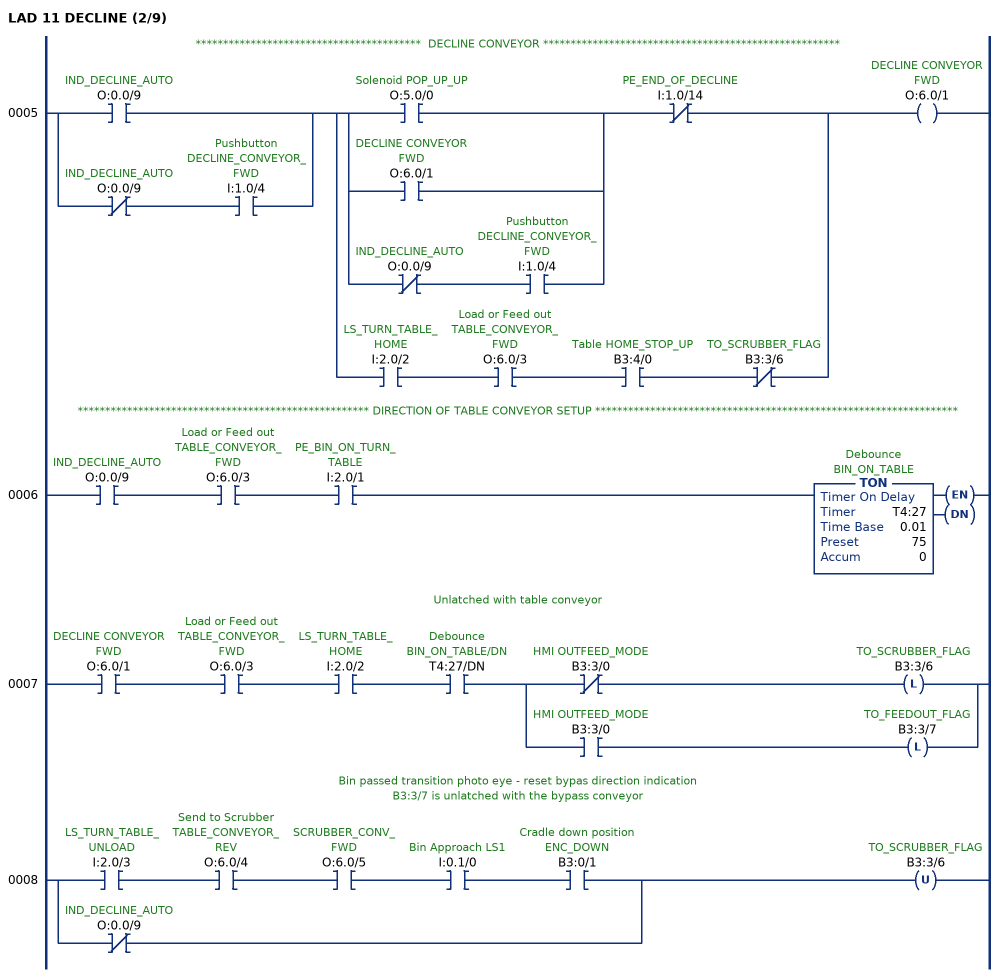
% Rung: 5 %
% *****************************************  DECLINE CONVEYOR ****************************************************** %
SOR BST XIC O:0.0/9 NXB XIO O:0.0/9 XIC I:1.0/4 BND BST BST XIC O:5.0/0 NXB BST XIC O:6.0/1 NXB XIO O:0.0/9 XIC I:1.0/4 BND BND XIO I:1.0/14 NXB XIC I:2.0/2 XIC O:6.0/3 XIC B3:4/0 XIO B3:3/6 BND OTE O:6.0/1 EOR
%   O:0.0/9  IND_DECLINE_AUTO %
%   I:1.0/4  DECLINE_CONVEYOR_FWD  "Pushbutton" %
%   O:5.0/0  POP_UP_UP  "Solenoid" %
%   O:6.0/1  "DECLINE CONVEYOR FWD" %
%   I:1.0/14  PE_END_OF_DECLINE %
%   I:2.0/2  LS_TURN_TABLE_HOME %
%   O:6.0/3  TABLE_CONVEYOR_FWD  "Load or Feed out" %
%   B3:4/0  HOME_STOP_UP  "Table" %
%   B3:3/6  TO_SCRUBBER_FLAG %
% Rung: 6 %
% ***************************************************** DIRECTION OF TABLE CONVEYOR SETUP ****************************************************************** %
SOR XIC O:0.0/9 XIC O:6.0/3 XIC I:2.0/1 TON T4:27 0.01 75 0 EOR
%   O:0.0/9  IND_DECLINE_AUTO %
%   O:6.0/3  TABLE_CONVEYOR_FWD  "Load or Feed out" %
%   I:2.0/1  PE_BIN_ON_TURN_TABLE %
%   T4:27  BIN_ON_TABLE  "Debounce" %
% Rung: 7 %
% Unlatched with table conveyor %
SOR XIC O:6.0/1 XIC O:6.0/3 XIC I:2.0/2 XIC T4:27/DN BST XIO B3:3/0 OTL B3:3/6 NXB XIC B3:3/0 OTL B3:3/7 BND EOR
%   O:6.0/1  "DECLINE CONVEYOR FWD" %
%   O:6.0/3  TABLE_CONVEYOR_FWD  "Load or Feed out" %
%   I:2.0/2  LS_TURN_TABLE_HOME %
%   T4:27  BIN_ON_TABLE  "Debounce" %
%   B3:3/0  OUTFEED_MODE  "HMI" %
%   B3:3/6  TO_SCRUBBER_FLAG %
%   B3:3/7  TO_FEEDOUT_FLAG %
% Rung: 8 %
% Bin passed transition photo eye - reset bypas direction indication
% B3:3/7 is unlatched with the bypass conveyor %
SOR BST XIC I:2.0/3 XIC O:6.0/4 XIC O:6.0/5 XIC I:0.1/0 XIC B3:0/1 NXB XIO O:0.0/9 BND OTU B3:3/6 EOR
%   I:2.0/3  LS_TURN_TABLE_UNLOAD %
%   O:6.0/4  TABLE_CONVEYOR_REV  "Send to Scrubber" %
%   O:6.0/5  SCRUBBER_CONV_FWD %
%   I:0.1/0  LS1  "Bin Approach" %
%   B3:0/1  ENC_DOWN  "Cradle down position" %
%   O:0.0/9  IND_DECLINE_AUTO %
%   B3:3/6  TO_SCRUBBER_FLAG %

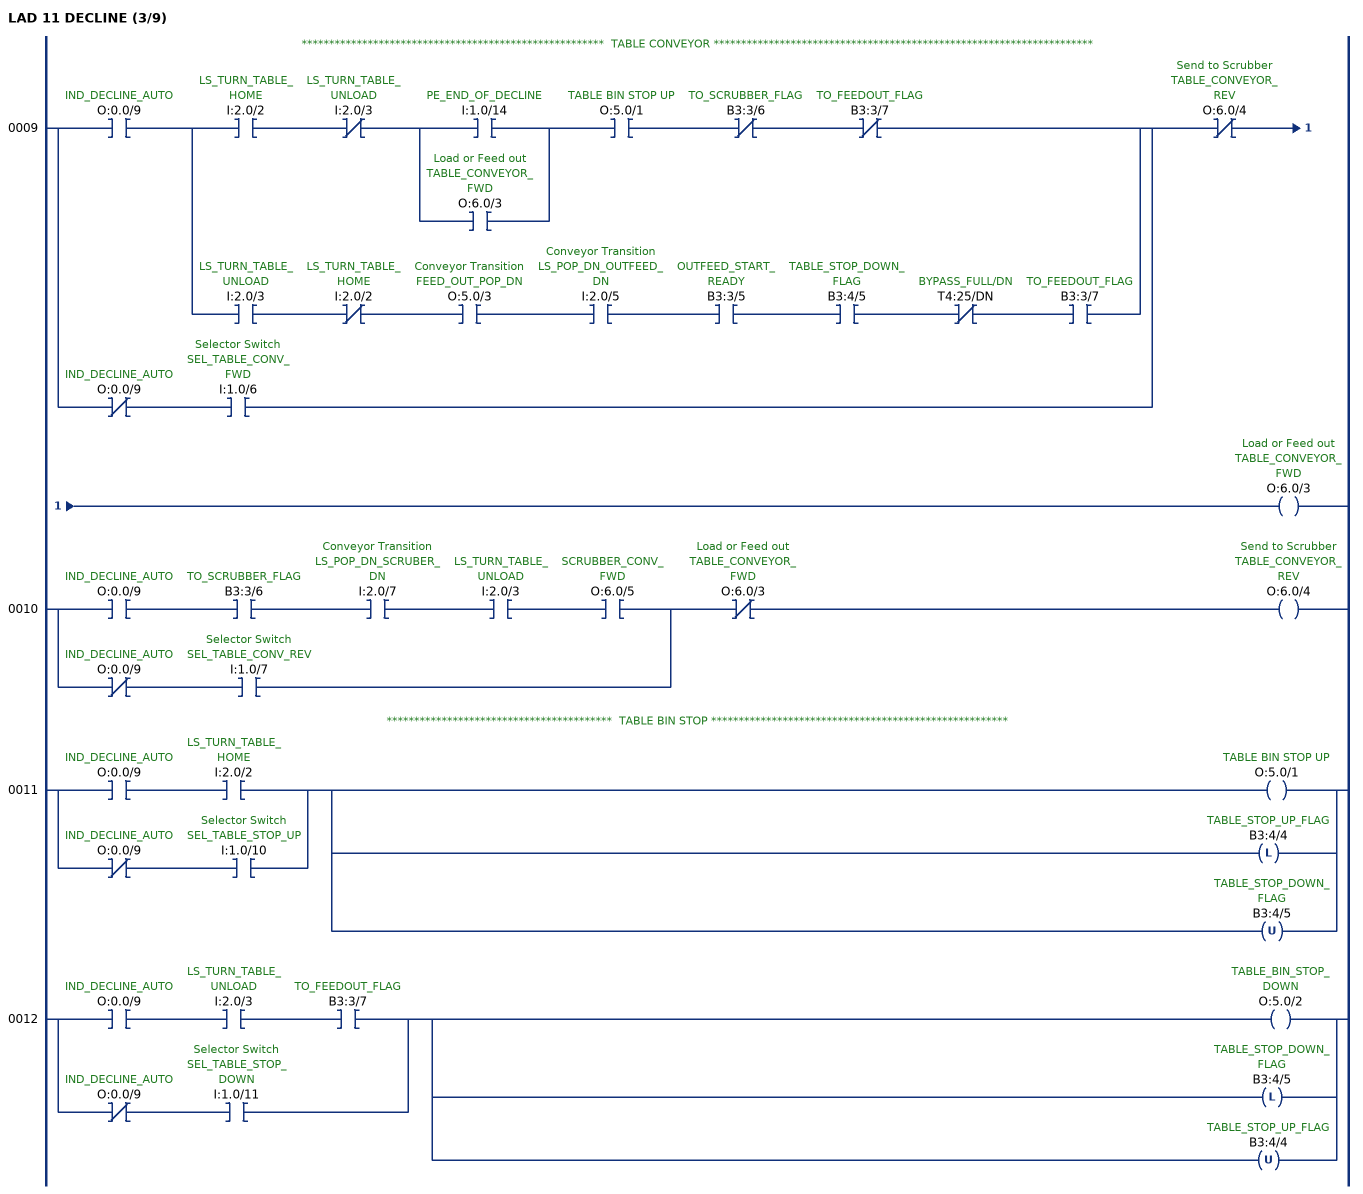
% Rung: 9 %
% *******************************************************  TABLE CONVEYOR ********************************************************************* %
SOR BST XIC O:0.0/9 BST XIC I:2.0/2 XIO I:2.0/3 BST XIC I:1.0/14 NXB XIC O:6.0/3 BND XIC O:5.0/1 XIO B3:3/6 XIO B3:3/7 NXB XIC I:2.0/3 XIO I:2.0/2 XIC O:5.0/3 XIC I:2.0/5 XIC B3:3/5 XIC B3:4/5 XIO T4:25/DN XIC B3:3/7 BND NXB XIO O:0.0/9 XIC I:1.0/6 BND XIO O:6.0/4 OTE O:6.0/3 EOR
%   O:0.0/9  IND_DECLINE_AUTO %
%   I:2.0/2  LS_TURN_TABLE_HOME %
%   I:2.0/3  LS_TURN_TABLE_UNLOAD %
%   I:1.0/14  PE_END_OF_DECLINE %
%   O:6.0/3  TABLE_CONVEYOR_FWD  "Load or Feed out" %
%   O:5.0/1  "TABLE BIN STOP UP" %
%   B3:3/6  TO_SCRUBBER_FLAG %
%   B3:3/7  TO_FEEDOUT_FLAG %
%   O:5.0/3  FEED_OUT_POP_DN  "Conveyor Transition" %
%   I:2.0/5  LS_POP_DN_OUTFEED_DN  "Conveyor Transition" %
%   B3:3/5  OUTFEED_START_READY %
%   B3:4/5  TABLE_STOP_DOWN_FLAG %
%   T4:25  BYPASS_FULL %
%   I:1.0/6  SEL_TABLE_CONV_FWD  "Selector Switch" %
%   O:6.0/4  TABLE_CONVEYOR_REV  "Send to Scrubber" %
% Rung: 10 %
SOR BST XIC O:0.0/9 XIC B3:3/6 XIC I:2.0/7 XIC I:2.0/3 XIC O:6.0/5 NXB XIO O:0.0/9 XIC I:1.0/7 BND XIO O:6.0/3 OTE O:6.0/4 EOR
%   O:0.0/9  IND_DECLINE_AUTO %
%   B3:3/6  TO_SCRUBBER_FLAG %
%   I:2.0/7  LS_POP_DN_SCRUBER_DN  "Conveyor Transition" %
%   I:2.0/3  LS_TURN_TABLE_UNLOAD %
%   O:6.0/5  SCRUBBER_CONV_FWD %
%   I:1.0/7  SEL_TABLE_CONV_REV  "Selector Switch" %
%   O:6.0/3  TABLE_CONVEYOR_FWD  "Load or Feed out" %
%   O:6.0/4  TABLE_CONVEYOR_REV  "Send to Scrubber" %
% Rung: 11 %
% *****************************************  TABLE BIN STOP ****************************************************** %
SOR BST XIC O:0.0/9 XIC I:2.0/2 NXB XIO O:0.0/9 XIC I:1.0/10 BND BST OTE O:5.0/1 NXB BST OTL B3:4/4 NXB OTU B3:4/5 BND BND EOR
%   O:0.0/9  IND_DECLINE_AUTO %
%   I:2.0/2  LS_TURN_TABLE_HOME %
%   I:1.0/10  SEL_TABLE_STOP_UP  "Selector Switch" %
%   O:5.0/1  "TABLE BIN STOP UP" %
%   B3:4/4  TABLE_STOP_UP_FLAG %
%   B3:4/5  TABLE_STOP_DOWN_FLAG %
% Rung: 12 %
SOR BST XIC O:0.0/9 XIC I:2.0/3 XIC B3:3/7 NXB XIO O:0.0/9 XIC I:1.0/11 BND BST OTE O:5.0/2 NXB BST OTL B3:4/5 NXB OTU B3:4/4 BND BND EOR
%   O:0.0/9  IND_DECLINE_AUTO %
%   I:2.0/3  LS_TURN_TABLE_UNLOAD %
%   B3:3/7  TO_FEEDOUT_FLAG %
%   I:1.0/11  SEL_TABLE_STOP_DOWN  "Selector Switch" %
%   O:5.0/2  "TABLE_BIN_STOP_DOWN" %
%   B3:4/5  TABLE_STOP_DOWN_FLAG %
%   B3:4/4  TABLE_STOP_UP_FLAG %

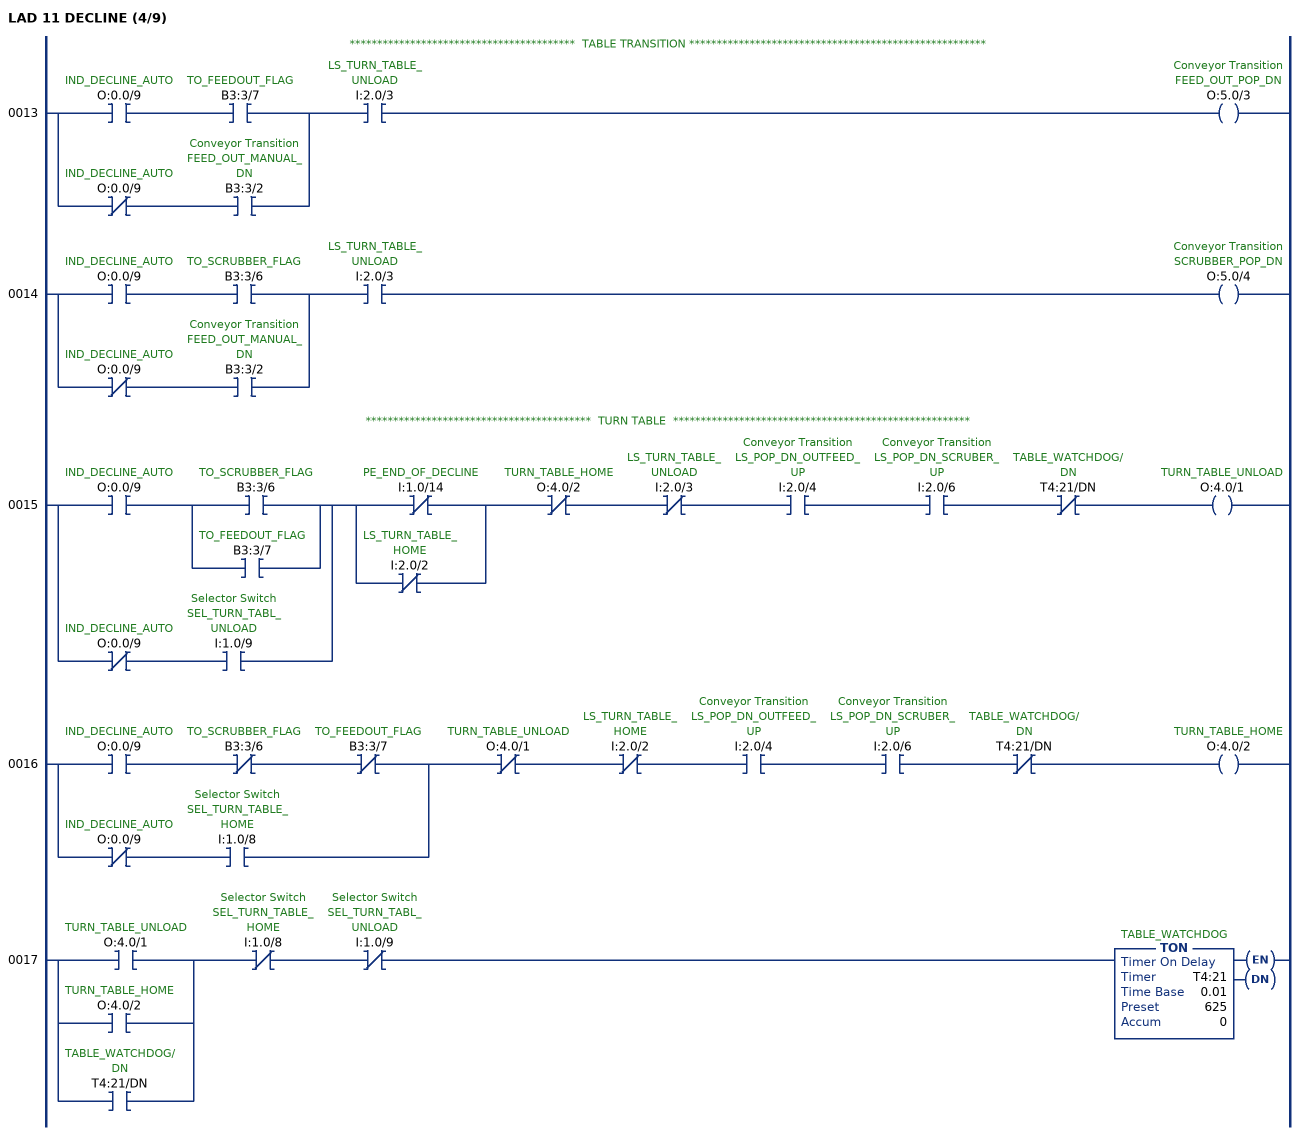
% Rung: 13 %
% *****************************************  TABLE TRANSITION ****************************************************** %
SOR BST XIC O:0.0/9 XIC B3:3/7 NXB XIO O:0.0/9 XIC B3:3/2 BND XIC I:2.0/3 OTE O:5.0/3 EOR
%   O:0.0/9  IND_DECLINE_AUTO %
%   B3:3/7  TO_FEEDOUT_FLAG %
%   B3:3/2  FEED_OUT_MANUAL_DN  "Conveyor Transition" %
%   I:2.0/3  LS_TURN_TABLE_UNLOAD %
%   O:5.0/3  FEED_OUT_POP_DN  "Conveyor Transition" %
% Rung: 14 %
SOR BST XIC O:0.0/9 XIC B3:3/6 NXB XIO O:0.0/9 XIC B3:3/2 BND XIC I:2.0/3 OTE O:5.0/4 EOR
%   O:0.0/9  IND_DECLINE_AUTO %
%   B3:3/6  TO_SCRUBBER_FLAG %
%   B3:3/2  FEED_OUT_MANUAL_DN  "Conveyor Transition" %
%   I:2.0/3  LS_TURN_TABLE_UNLOAD %
%   O:5.0/4  SCRUBBER_POP_DN  "Conveyor Transition" %
% Rung: 15 %
% *****************************************  TURN TABLE  ****************************************************** %
SOR BST XIC O:0.0/9 BST XIC B3:3/6 NXB XIC B3:3/7 BND NXB XIO O:0.0/9 XIC I:1.0/9 BND BST XIO I:1.0/14 NXB XIO I:2.0/2 BND XIO O:4.0/2 XIO I:2.0/3 XIC I:2.0/4 XIC I:2.0/6 XIO T4:21/DN OTE O:4.0/1 EOR
%   O:0.0/9  IND_DECLINE_AUTO %
%   B3:3/6  TO_SCRUBBER_FLAG %
%   B3:3/7  TO_FEEDOUT_FLAG %
%   I:1.0/9  SEL_TURN_TABL_UNLOAD  "Selector Switch" %
%   I:1.0/14  PE_END_OF_DECLINE %
%   I:2.0/2  LS_TURN_TABLE_HOME %
%   O:4.0/2  TURN_TABLE_HOME %
%   I:2.0/3  LS_TURN_TABLE_UNLOAD %
%   I:2.0/4  LS_POP_DN_OUTFEED_UP  "Conveyor Transition" %
%   I:2.0/6  LS_POP_DN_SCRUBER_UP  "Conveyor Transition" %
%   T4:21  TABLE_WATCHDOG %
%   O:4.0/1  TURN_TABLE_UNLOAD %
% Rung: 16 %
SOR BST XIC O:0.0/9 XIO B3:3/6 XIO B3:3/7 NXB XIO O:0.0/9 XIC I:1.0/8 BND XIO O:4.0/1 XIO I:2.0/2 XIC I:2.0/4 XIC I:2.0/6 XIO T4:21/DN OTE O:4.0/2 EOR
%   O:0.0/9  IND_DECLINE_AUTO %
%   B3:3/6  TO_SCRUBBER_FLAG %
%   B3:3/7  TO_FEEDOUT_FLAG %
%   I:1.0/8  SEL_TURN_TABLE_HOME  "Selector Switch" %
%   O:4.0/1  TURN_TABLE_UNLOAD %
%   I:2.0/2  LS_TURN_TABLE_HOME %
%   I:2.0/4  LS_POP_DN_OUTFEED_UP  "Conveyor Transition" %
%   I:2.0/6  LS_POP_DN_SCRUBER_UP  "Conveyor Transition" %
%   T4:21  TABLE_WATCHDOG %
%   O:4.0/2  TURN_TABLE_HOME %
% Rung: 17 %
SOR BST BST XIC O:4.0/1 NXB XIC O:4.0/2 BND NXB XIC T4:21/DN BND XIO I:1.0/8 XIO I:1.0/9 TON T4:21 0.01 625 0 EOR
%   O:4.0/1  TURN_TABLE_UNLOAD %
%   O:4.0/2  TURN_TABLE_HOME %
%   T4:21  TABLE_WATCHDOG %
%   I:1.0/8  SEL_TURN_TABLE_HOME  "Selector Switch" %
%   I:1.0/9  SEL_TURN_TABL_UNLOAD  "Selector Switch" %

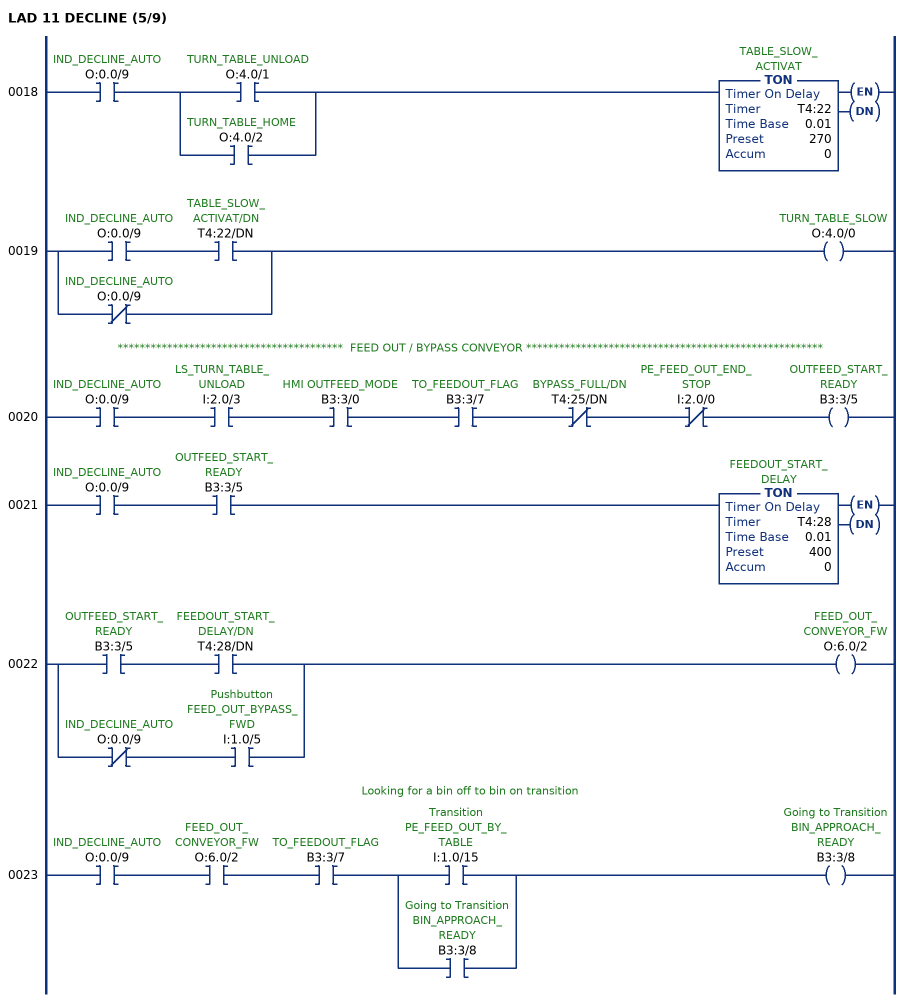
% Rung: 18 %
SOR XIC O:0.0/9 BST XIC O:4.0/1 NXB XIC O:4.0/2 BND TON T4:22 0.01 270 0 EOR
%   O:0.0/9  IND_DECLINE_AUTO %
%   O:4.0/1  TURN_TABLE_UNLOAD %
%   O:4.0/2  TURN_TABLE_HOME %
%   T4:22  TABLE_SLOW_ACTIVAT %
% Rung: 19 %
SOR BST XIC O:0.0/9 XIC T4:22/DN NXB XIO O:0.0/9 BND OTE O:4.0/0 EOR
%   O:0.0/9  IND_DECLINE_AUTO %
%   T4:22  TABLE_SLOW_ACTIVAT %
%   O:4.0/0  TURN_TABLE_SLOW %
% Rung: 20 %
% *****************************************  FEED OUT / BYPASS CONVEYOR ****************************************************** %
SOR XIC O:0.0/9 XIC I:2.0/3 XIC B3:3/0 XIC B3:3/7 XIO T4:25/DN XIO I:2.0/0 OTE B3:3/5 EOR
%   O:0.0/9  IND_DECLINE_AUTO %
%   I:2.0/3  LS_TURN_TABLE_UNLOAD %
%   B3:3/0  OUTFEED_MODE  "HMI" %
%   B3:3/7  TO_FEEDOUT_FLAG %
%   T4:25  BYPASS_FULL %
%   I:2.0/0  PE_FEED_OUT_END_STOP %
%   B3:3/5  OUTFEED_START_READY %
% Rung: 21 %
SOR XIC O:0.0/9 XIC B3:3/5 TON T4:28 0.01 400 0 EOR
%   O:0.0/9  IND_DECLINE_AUTO %
%   B3:3/5  OUTFEED_START_READY %
%   T4:28  FEEDOUT_START_DELAY %
% Rung: 22 %
SOR BST XIC B3:3/5 XIC T4:28/DN NXB XIO O:0.0/9 XIC I:1.0/5 BND OTE O:6.0/2 EOR
%   B3:3/5  OUTFEED_START_READY %
%   T4:28  FEEDOUT_START_DELAY %
%   O:0.0/9  IND_DECLINE_AUTO %
%   I:1.0/5  FEED_OUT_BYPASS_FWD  "Pushbutton" %
%   O:6.0/2  FEED_OUT_CONVEYOR_FW %
% Rung: 23 %
% Looking for a bin off to bin on transition %
SOR XIC O:0.0/9 XIC O:6.0/2 XIC B3:3/7 BST XIC I:1.0/15 NXB XIC B3:3/8 BND OTE B3:3/8 EOR
%   O:0.0/9  IND_DECLINE_AUTO %
%   O:6.0/2  FEED_OUT_CONVEYOR_FW %
%   B3:3/7  TO_FEEDOUT_FLAG %
%   I:1.0/15  PE_FEED_OUT_BY_TABLE  "Transition" %
%   B3:3/8  BIN_APPROACH_READY  "Going to Transition" %

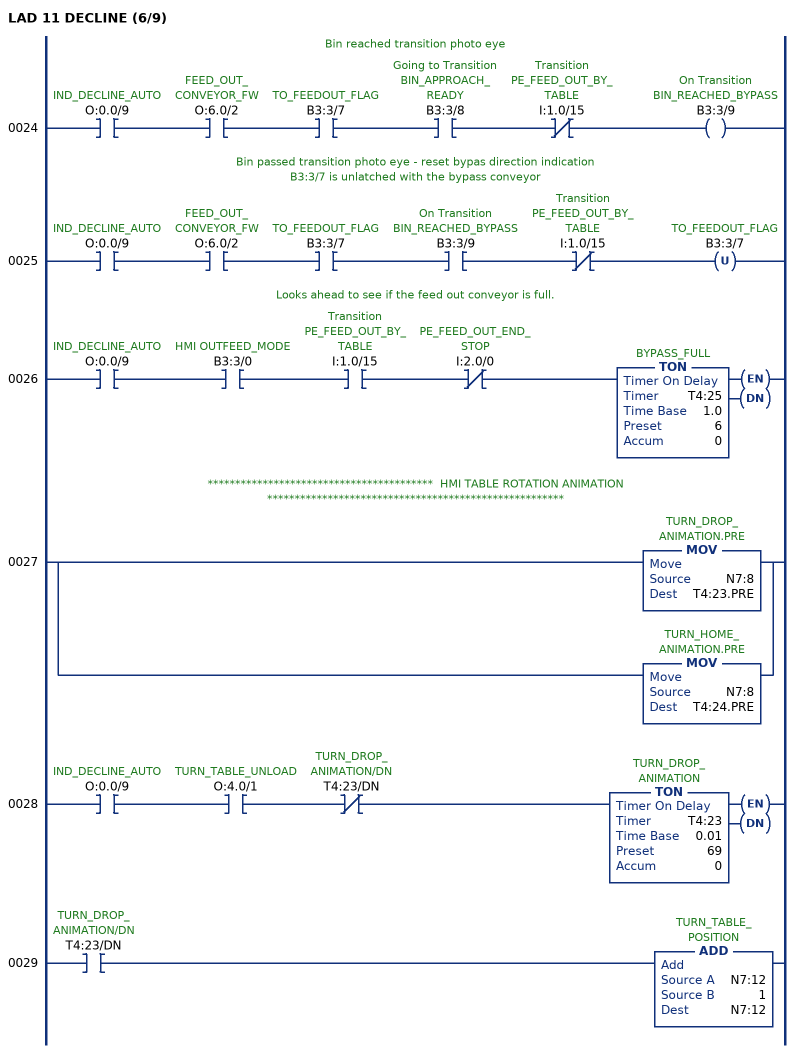
% Rung: 24 %
% Bin reached transition photo eye %
SOR XIC O:0.0/9 XIC O:6.0/2 XIC B3:3/7 XIC B3:3/8 XIO I:1.0/15 OTE B3:3/9 EOR
%   O:0.0/9  IND_DECLINE_AUTO %
%   O:6.0/2  FEED_OUT_CONVEYOR_FW %
%   B3:3/7  TO_FEEDOUT_FLAG %
%   B3:3/8  BIN_APPROACH_READY  "Going to Transition" %
%   I:1.0/15  PE_FEED_OUT_BY_TABLE  "Transition" %
%   B3:3/9  BIN_REACHED_BYPASS  "On Transition" %
% Rung: 25 %
% Bin passed transition photo eye - reset bypas direction indication
% B3:3/7 is unlatched with the bypass conveyor %
SOR XIC O:0.0/9 XIC O:6.0/2 XIC B3:3/7 XIC B3:3/9 XIO I:1.0/15 OTU B3:3/7 EOR
%   O:0.0/9  IND_DECLINE_AUTO %
%   O:6.0/2  FEED_OUT_CONVEYOR_FW %
%   B3:3/7  TO_FEEDOUT_FLAG %
%   B3:3/9  BIN_REACHED_BYPASS  "On Transition" %
%   I:1.0/15  PE_FEED_OUT_BY_TABLE  "Transition" %
% Rung: 26 %
% Looks ahead to see if the feed out conveyor is full. %
SOR XIC O:0.0/9 XIC B3:3/0 XIC I:1.0/15 XIO I:2.0/0 TON T4:25 1.0 6 0 EOR
%   O:0.0/9  IND_DECLINE_AUTO %
%   B3:3/0  OUTFEED_MODE  "HMI" %
%   I:1.0/15  PE_FEED_OUT_BY_TABLE  "Transition" %
%   I:2.0/0  PE_FEED_OUT_END_STOP %
%   T4:25  BYPASS_FULL %
% Rung: 27 %
% *****************************************  HMI TABLE ROTATION ANIMATION  ****************************************************** %
SOR BST MOV N7:8 T4:23.PRE NXB MOV N7:8 T4:24.PRE BND EOR
%   N7:8  TABLE_ANIMATION_TIME %
%   T4:23  TURN_DROP_ANIMATION %
%   T4:24  TURN_HOME_ANIMATION %
% Rung: 28 %
SOR XIC O:0.0/9 XIC O:4.0/1 XIO T4:23/DN TON T4:23 0.01 69 0 EOR
%   O:0.0/9  IND_DECLINE_AUTO %
%   O:4.0/1  TURN_TABLE_UNLOAD %
%   T4:23  TURN_DROP_ANIMATION %
% Rung: 29 %
SOR XIC T4:23/DN ADD N7:12 1 N7:12 EOR
%   T4:23  TURN_DROP_ANIMATION %
%   N7:12  TURN_TABLE_POSITION %

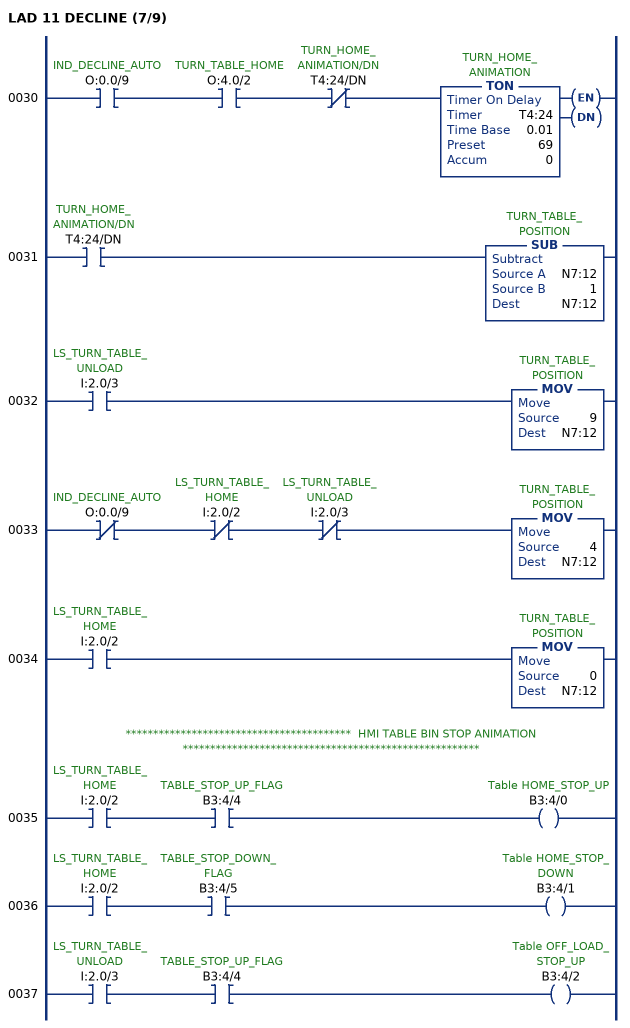
% Rung: 30 %
SOR XIC O:0.0/9 XIC O:4.0/2 XIO T4:24/DN TON T4:24 0.01 69 0 EOR
%   O:0.0/9  IND_DECLINE_AUTO %
%   O:4.0/2  TURN_TABLE_HOME %
%   T4:24  TURN_HOME_ANIMATION %
% Rung: 31 %
SOR XIC T4:24/DN SUB N7:12 1 N7:12 EOR
%   T4:24  TURN_HOME_ANIMATION %
%   N7:12  TURN_TABLE_POSITION %
% Rung: 32 %
SOR XIC I:2.0/3 MOV 9 N7:12 EOR
%   I:2.0/3  LS_TURN_TABLE_UNLOAD %
%   N7:12  TURN_TABLE_POSITION %
% Rung: 33 %
SOR XIO O:0.0/9 XIO I:2.0/2 XIO I:2.0/3 MOV 4 N7:12 EOR
%   O:0.0/9  IND_DECLINE_AUTO %
%   I:2.0/2  LS_TURN_TABLE_HOME %
%   I:2.0/3  LS_TURN_TABLE_UNLOAD %
%   N7:12  TURN_TABLE_POSITION %
% Rung: 34 %
SOR XIC I:2.0/2 MOV 0 N7:12 EOR
%   I:2.0/2  LS_TURN_TABLE_HOME %
%   N7:12  TURN_TABLE_POSITION %
% Rung: 35 %
% *****************************************  HMI TABLE BIN STOP ANIMATION  ****************************************************** %
SOR XIC I:2.0/2 XIC B3:4/4 OTE B3:4/0 EOR
%   I:2.0/2  LS_TURN_TABLE_HOME %
%   B3:4/4  TABLE_STOP_UP_FLAG %
%   B3:4/0  HOME_STOP_UP  "Table" %
% Rung: 36 %
SOR XIC I:2.0/2 XIC B3:4/5 OTE B3:4/1 EOR
%   I:2.0/2  LS_TURN_TABLE_HOME %
%   B3:4/5  TABLE_STOP_DOWN_FLAG %
%   B3:4/1  HOME_STOP_DOWN  "Table" %
% Rung: 37 %
SOR XIC I:2.0/3 XIC B3:4/4 OTE B3:4/2 EOR
%   I:2.0/3  LS_TURN_TABLE_UNLOAD %
%   B3:4/4  TABLE_STOP_UP_FLAG %
%   B3:4/2  OFF_LOAD_STOP_UP  "Table" %

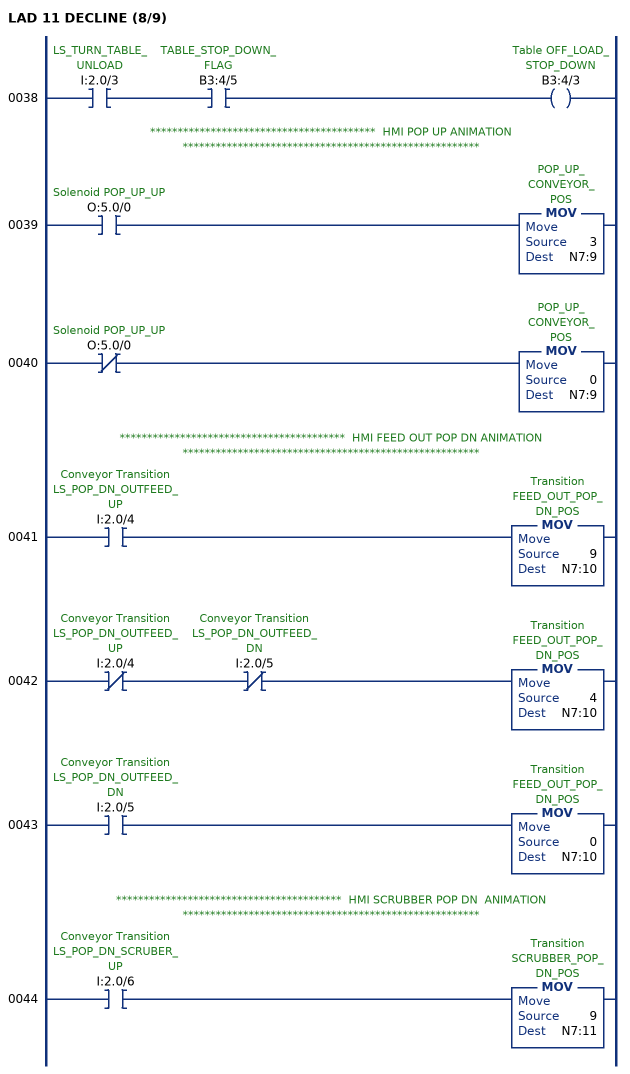
% Rung: 38 %
SOR XIC I:2.0/3 XIC B3:4/5 OTE B3:4/3 EOR
%   I:2.0/3  LS_TURN_TABLE_UNLOAD %
%   B3:4/5  TABLE_STOP_DOWN_FLAG %
%   B3:4/3  OFF_LOAD_STOP_DOWN  "Table" %
% Rung: 39 %
% *****************************************  HMI POP UP ANIMATION  ****************************************************** %
SOR XIC O:5.0/0 MOV 3 N7:9 EOR
%   O:5.0/0  POP_UP_UP  "Solenoid" %
%   N7:9  POP_UP_CONVEYOR_POS %
% Rung: 40 %
SOR XIO O:5.0/0 MOV 0 N7:9 EOR
%   O:5.0/0  POP_UP_UP  "Solenoid" %
%   N7:9  POP_UP_CONVEYOR_POS %
% Rung: 41 %
% *****************************************  HMI FEED OUT POP DN ANIMATION  ****************************************************** %
SOR XIC I:2.0/4 MOV 9 N7:10 EOR
%   I:2.0/4  LS_POP_DN_OUTFEED_UP  "Conveyor Transition" %
%   N7:10  FEED_OUT_POP_DN_POS  "Transition" %
% Rung: 42 %
SOR XIO I:2.0/4 XIO I:2.0/5 MOV 4 N7:10 EOR
%   I:2.0/4  LS_POP_DN_OUTFEED_UP  "Conveyor Transition" %
%   I:2.0/5  LS_POP_DN_OUTFEED_DN  "Conveyor Transition" %
%   N7:10  FEED_OUT_POP_DN_POS  "Transition" %
% Rung: 43 %
SOR XIC I:2.0/5 MOV 0 N7:10 EOR
%   I:2.0/5  LS_POP_DN_OUTFEED_DN  "Conveyor Transition" %
%   N7:10  FEED_OUT_POP_DN_POS  "Transition" %
% Rung: 44 %
% *****************************************  HMI SCRUBBER POP DN  ANIMATION  ****************************************************** %
SOR XIC I:2.0/6 MOV 9 N7:11 EOR
%   I:2.0/6  LS_POP_DN_SCRUBER_UP  "Conveyor Transition" %
%   N7:11  SCRUBBER_POP_DN_POS  "Transition" %

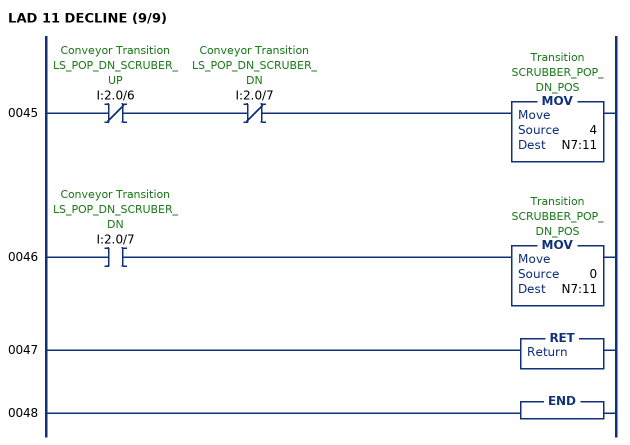
% Rung: 45 %
SOR XIO I:2.0/6 XIO I:2.0/7 MOV 4 N7:11 EOR
%   I:2.0/6  LS_POP_DN_SCRUBER_UP  "Conveyor Transition" %
%   I:2.0/7  LS_POP_DN_SCRUBER_DN  "Conveyor Transition" %
%   N7:11  SCRUBBER_POP_DN_POS  "Transition" %
% Rung: 46 %
SOR XIC I:2.0/7 MOV 0 N7:11 EOR
%   I:2.0/7  LS_POP_DN_SCRUBER_DN  "Conveyor Transition" %
%   N7:11  SCRUBBER_POP_DN_POS  "Transition" %
% Rung: 47 %
SOR RET EOR
% Rung: 48 %
SOR END EOR

LADDER 12 "STACK LS"
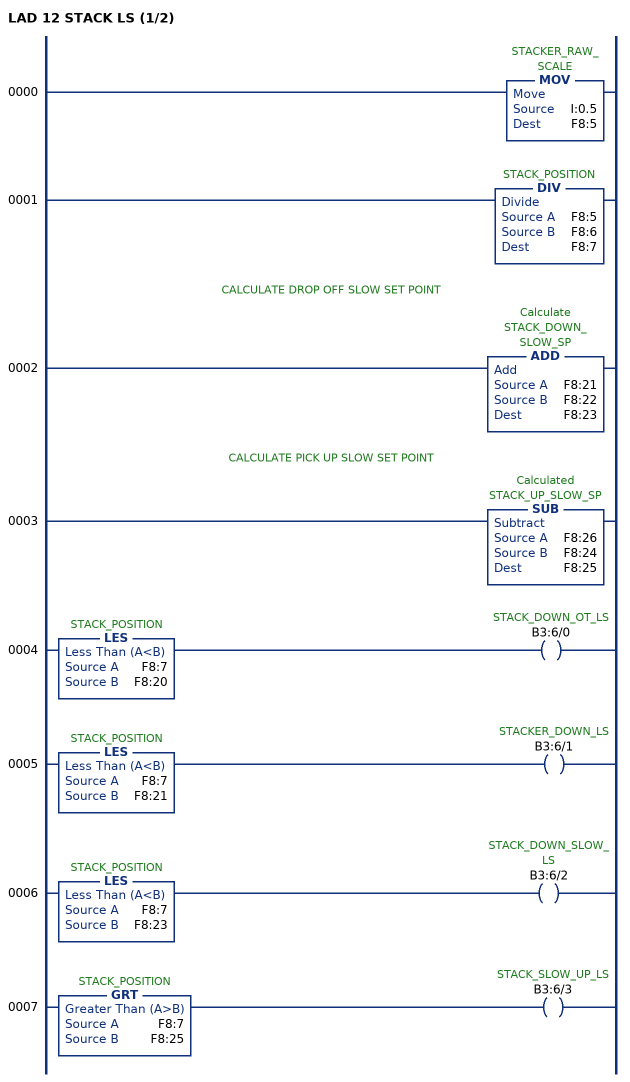
% Rung: 0 %
SOR MOV I:0.5 F8:5 EOR
%   F8:5  STACKER_RAW_SCALE %
% Rung: 1 %
SOR DIV F8:5 F8:6 F8:7 EOR
%   F8:5  STACKER_RAW_SCALE %
%   F8:6  STACK_SCALLER %
%   F8:7  STACK_POSITION %
% Rung: 2 %
% CALCULATE DROP OFF SLOW SET POINT %
SOR ADD F8:21 F8:22 F8:23 EOR
%   F8:21  RESTACK_DOWN_SP  "Actual" %
%   F8:22  RESTACK_DOWN_SLOW  "Offset" %
%   F8:23  STACK_DOWN_SLOW_SP  "Calculate" %
% Rung: 3 %
% CALCULATE PICK UP SLOW SET POINT %
SOR SUB F8:26 F8:24 F8:25 EOR
%   F8:26  RESTACK_UP_SP %
%   F8:24  RESTACK_SLOW_UP  "Offset" %
%   F8:25  STACK_UP_SLOW_SP  "Calculated" %
% Rung: 4 %
SOR LES F8:7 F8:20 OTE B3:6/0 EOR
%   F8:7  STACK_POSITION %
%   F8:20  RESTACK_DOWN_OT_SP %
%   B3:6/0  STACK_DOWN_OT_LS %
% Rung: 5 %
SOR LES F8:7 F8:21 OTE B3:6/1 EOR
%   F8:7  STACK_POSITION %
%   F8:21  RESTACK_DOWN_SP  "Actual" %
%   B3:6/1  STACKER_DOWN_LS %
% Rung: 6 %
SOR LES F8:7 F8:23 OTE B3:6/2 EOR
%   F8:7  STACK_POSITION %
%   F8:23  STACK_DOWN_SLOW_SP  "Calculate" %
%   B3:6/2  STACK_DOWN_SLOW_LS %
% Rung: 7 %
SOR GRT F8:7 F8:25 OTE B3:6/3 EOR
%   F8:7  STACK_POSITION %
%   F8:25  STACK_UP_SLOW_SP  "Calculated" %
%   B3:6/3  STACK_SLOW_UP_LS %

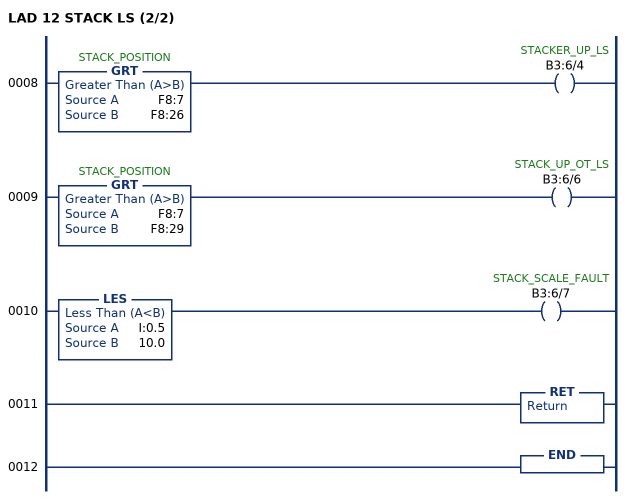
% Rung: 8 %
SOR GRT F8:7 F8:26 OTE B3:6/4 EOR
%   F8:7  STACK_POSITION %
%   F8:26  RESTACK_UP_SP %
%   B3:6/4  STACKER_UP_LS %
% Rung: 9 %
SOR GRT F8:7 F8:29 OTE B3:6/6 EOR
%   F8:7  STACK_POSITION %
%   F8:29  RESTACK_UP_OT_SP  "Actual" %
%   B3:6/6  STACK_UP_OT_LS %
% Rung: 10 %
SOR LES I:0.5 10.0 OTE B3:6/7 EOR
%   B3:6/7  STACK_SCALE_FAULT %
% Rung: 11 %
SOR RET EOR
% Rung: 12 %
SOR END EOR

LADDER 13 "STACK"
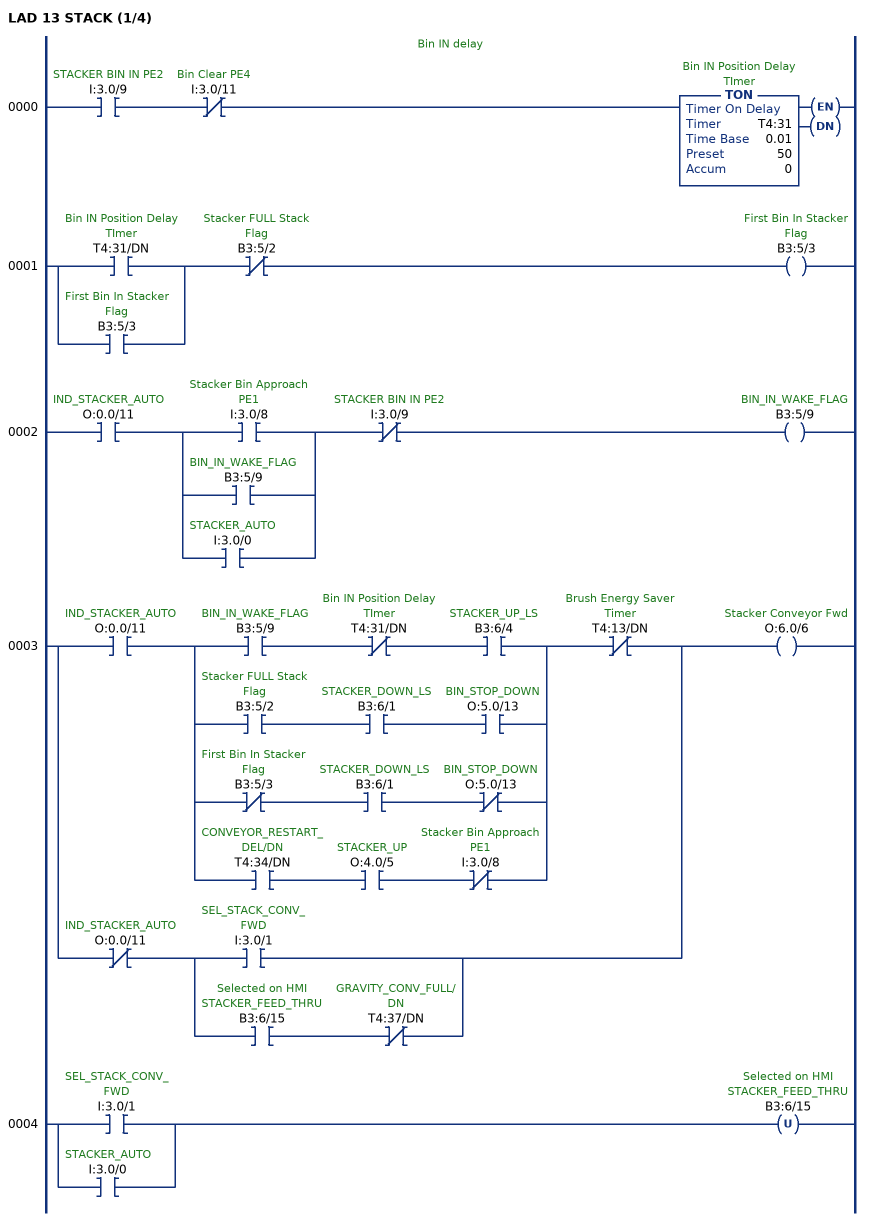
% Rung: 0 %
% Bin IN delay %
SOR XIC I:3.0/9 XIO I:3.0/11 TON T4:31 0.01 50 0 EOR
%   I:3.0/9  PE2  "STACKER BIN IN" %
%   I:3.0/11  PE4  "Bin Clear" %
%   T4:31  "Bin IN Position Delay TImer" %
% Rung: 1 %
SOR BST XIC T4:31/DN NXB XIC B3:5/3 BND XIO B3:5/2 OTE B3:5/3 EOR
%   T4:31  "Bin IN Position Delay TImer" %
%   B3:5/3  "First Bin In Stacker Flag" %
%   B3:5/2  "Stacker FULL Stack Flag" %
% Rung: 2 %
SOR XIC O:0.0/11 BST XIC I:3.0/8 NXB BST XIC B3:5/9 NXB XIC I:3.0/0 BND BND XIO I:3.0/9 OTE B3:5/9 EOR
%   O:0.0/11  IND_STACKER_AUTO %
%   I:3.0/8  PE1  "Stacker Bin Approach" %
%   B3:5/9  BIN_IN_WAKE_FLAG %
%   I:3.0/0  STACKER_AUTO %
%   I:3.0/9  PE2  "STACKER BIN IN" %
% Rung: 3 %
SOR BST XIC O:0.0/11 BST XIC B3:5/9 XIO T4:31/DN XIC B3:6/4 NXB XIC B3:5/2 XIC B3:6/1 XIC O:5.0/13 NXB BST XIO B3:5/3 XIC B3:6/1 XIO O:5.0/13 NXB XIC T4:34/DN XIC O:4.0/5 XIO I:3.0/8 BND BND XIO T4:13/DN NXB XIO O:0.0/11 BST XIC I:3.0/1 NXB XIC B3:6/15 XIO T4:37/DN BND BND OTE O:6.0/6 EOR
%   O:0.0/11  IND_STACKER_AUTO %
%   B3:5/9  BIN_IN_WAKE_FLAG %
%   T4:31  "Bin IN Position Delay TImer" %
%   B3:6/4  STACKER_UP_LS %
%   B3:5/2  "Stacker FULL Stack Flag" %
%   B3:6/1  STACKER_DOWN_LS %
%   O:5.0/13  BIN_STOP_DOWN %
%   B3:5/3  "First Bin In Stacker Flag" %
%   T4:34  CONVEYOR_RESTART_DEL %
%   O:4.0/5  STACKER_UP %
%   I:3.0/8  PE1  "Stacker Bin Approach" %
%   T4:13  "Brush Energy Saver Timer" %
%   I:3.0/1  SEL_STACK_CONV_FWD %
%   B3:6/15  STACKER_FEED_THRU  "Selected on HMI" %
%   T4:37  GRAVITY_CONV_FULL %
%   O:6.0/6  "Stacker Conveyor Fwd" %
% Rung: 4 %
SOR BST XIC I:3.0/1 NXB XIC I:3.0/0 BND OTU B3:6/15 EOR
%   I:3.0/1  SEL_STACK_CONV_FWD %
%   I:3.0/0  STACKER_AUTO %
%   B3:6/15  STACKER_FEED_THRU  "Selected on HMI" %

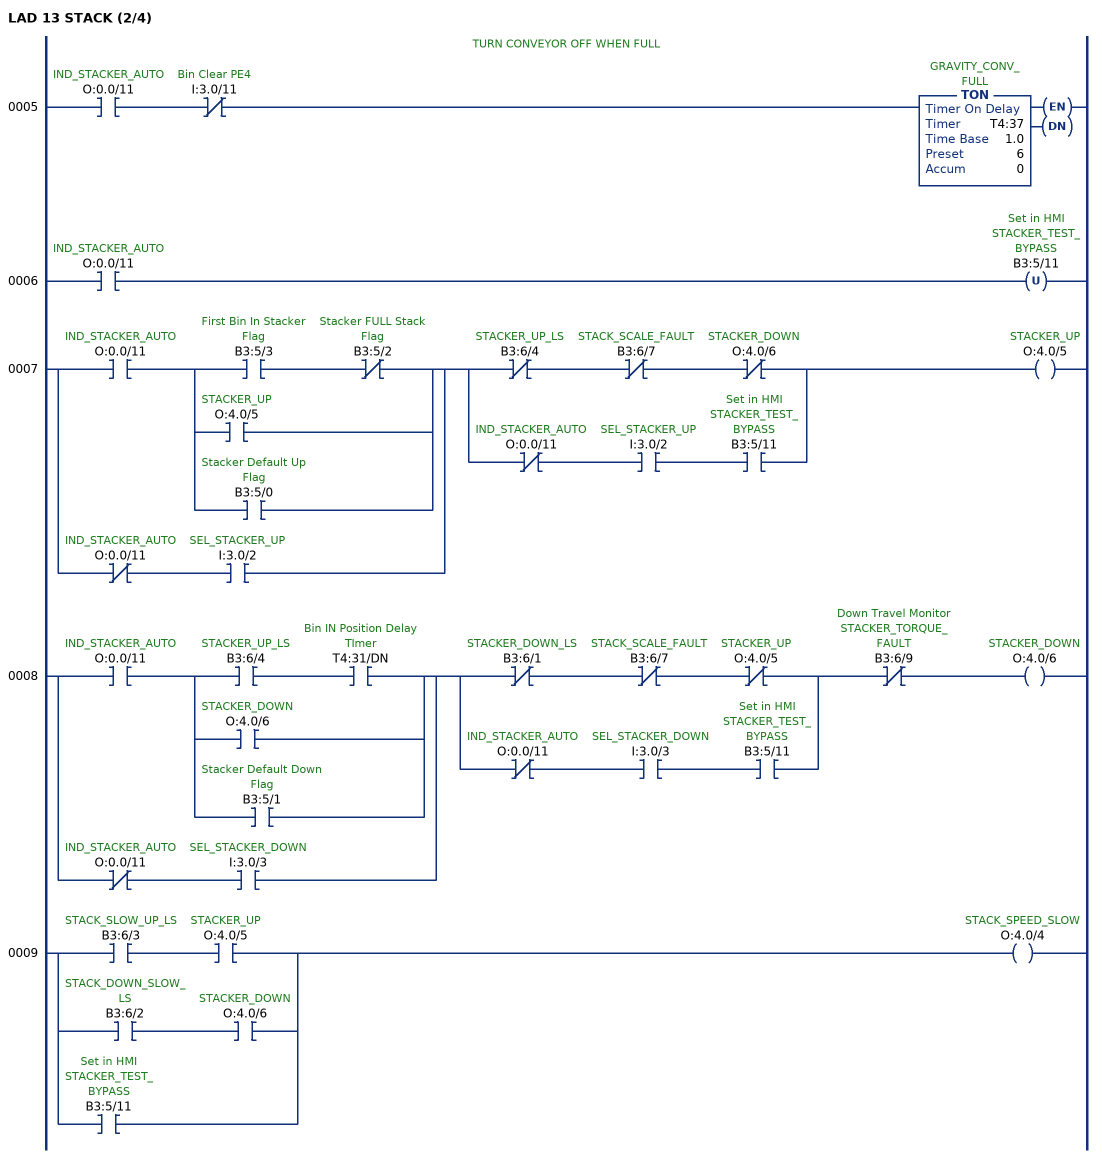
% Rung: 5 %
% TURN CONVEYOR OFF WHEN FULL %
SOR XIC O:0.0/11 XIO I:3.0/11 TON T4:37 1.0 6 0 EOR
%   O:0.0/11  IND_STACKER_AUTO %
%   I:3.0/11  PE4  "Bin Clear" %
%   T4:37  GRAVITY_CONV_FULL %
% Rung: 6 %
SOR XIC O:0.0/11 OTU B3:5/11 EOR
%   O:0.0/11  IND_STACKER_AUTO %
%   B3:5/11  STACKER_TEST_BYPASS  "Set in HMI" %
% Rung: 7 %
SOR BST XIC O:0.0/11 BST XIC B3:5/3 XIO B3:5/2 NXB XIC O:4.0/5 NXB XIC B3:5/0 BND NXB XIO O:0.0/11 XIC I:3.0/2 BND BST XIO B3:6/4 XIO B3:6/7 XIO O:4.0/6 NXB XIO O:0.0/11 XIC I:3.0/2 XIC B3:5/11 BND OTE O:4.0/5 EOR
%   O:0.0/11  IND_STACKER_AUTO %
%   B3:5/3  "First Bin In Stacker Flag" %
%   B3:5/2  "Stacker FULL Stack Flag" %
%   O:4.0/5  STACKER_UP %
%   B3:5/0  "Stacker Default Up Flag" %
%   I:3.0/2  SEL_STACKER_UP %
%   B3:6/4  STACKER_UP_LS %
%   B3:6/7  STACK_SCALE_FAULT %
%   O:4.0/6  STACKER_DOWN %
%   B3:5/11  STACKER_TEST_BYPASS  "Set in HMI" %
% Rung: 8 %
SOR BST XIC O:0.0/11 BST XIC B3:6/4 XIC T4:31/DN NXB XIC O:4.0/6 NXB XIC B3:5/1 BND NXB XIO O:0.0/11 XIC I:3.0/3 BND BST XIO B3:6/1 XIO B3:6/7 XIO O:4.0/5 NXB XIO O:0.0/11 XIC I:3.0/3 XIC B3:5/11 BND XIO B3:6/9 OTE O:4.0/6 EOR
%   O:0.0/11  IND_STACKER_AUTO %
%   B3:6/4  STACKER_UP_LS %
%   T4:31  "Bin IN Position Delay TImer" %
%   O:4.0/6  STACKER_DOWN %
%   B3:5/1  "Stacker Default Down Flag" %
%   I:3.0/3  SEL_STACKER_DOWN %
%   B3:6/1  STACKER_DOWN_LS %
%   B3:6/7  STACK_SCALE_FAULT %
%   O:4.0/5  STACKER_UP %
%   B3:5/11  STACKER_TEST_BYPASS  "Set in HMI" %
%   B3:6/9  STACKER_TORQUE_FAULT  "Down Travel Monitor" %
% Rung: 9 %
SOR BST BST XIC B3:6/3 XIC O:4.0/5 NXB XIC B3:6/2 XIC O:4.0/6 BND NXB XIC B3:5/11 BND OTE O:4.0/4 EOR
%   B3:6/3  STACK_SLOW_UP_LS %
%   O:4.0/5  STACKER_UP %
%   B3:6/2  STACK_DOWN_SLOW_LS %
%   O:4.0/6  STACKER_DOWN %
%   B3:5/11  STACKER_TEST_BYPASS  "Set in HMI" %
%   O:4.0/4  STACK_SPEED_SLOW %

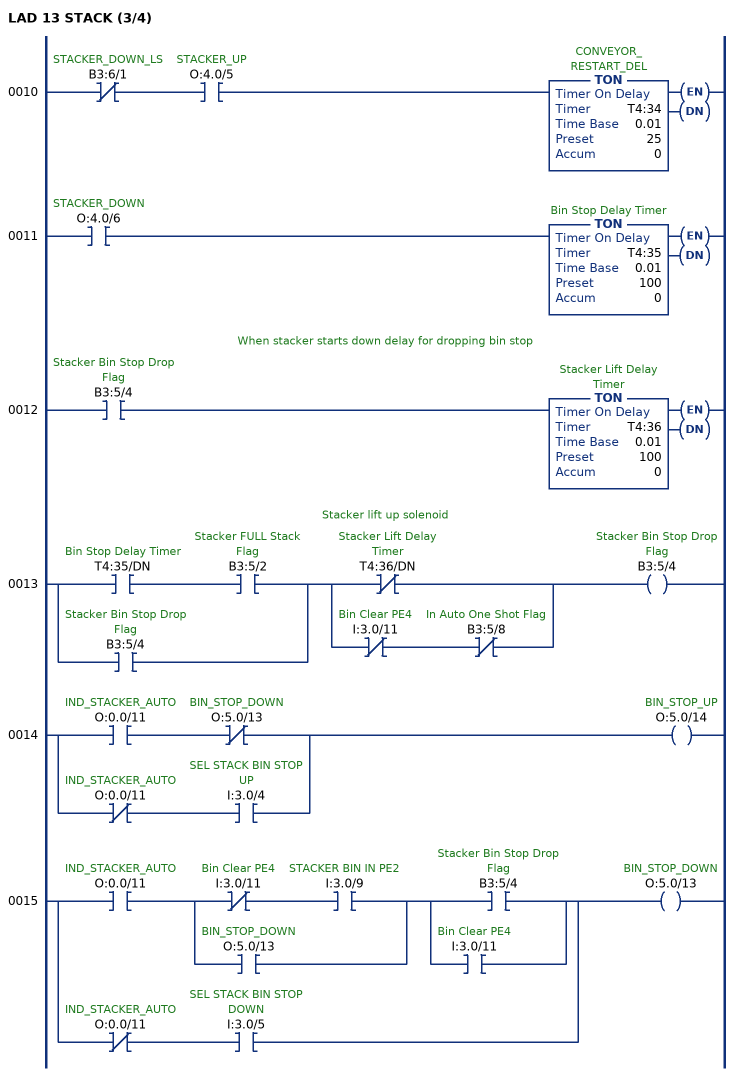
% Rung: 10 %
SOR XIO B3:6/1 XIC O:4.0/5 TON T4:34 0.01 25 0 EOR
%   B3:6/1  STACKER_DOWN_LS %
%   O:4.0/5  STACKER_UP %
%   T4:34  CONVEYOR_RESTART_DEL %
% Rung: 11 %
SOR XIC O:4.0/6 TON T4:35 0.01 100 0 EOR
%   O:4.0/6  STACKER_DOWN %
%   T4:35  "Bin Stop Delay Timer" %
% Rung: 12 %
% When stacker starts down delay for dropping bin stop %
SOR XIC B3:5/4 TON T4:36 0.01 100 0 EOR
%   B3:5/4  "Stacker Bin Stop Drop Flag" %
%   T4:36  "Stacker Lift Delay Timer" %
% Rung: 13 %
% Stacker lift up solenoid %
SOR BST XIC T4:35/DN XIC B3:5/2 NXB XIC B3:5/4 BND BST XIO T4:36/DN NXB XIO I:3.0/11 XIO B3:5/8 BND OTE B3:5/4 EOR
%   T4:35  "Bin Stop Delay Timer" %
%   B3:5/2  "Stacker FULL Stack Flag" %
%   B3:5/4  "Stacker Bin Stop Drop Flag" %
%   T4:36  "Stacker Lift Delay Timer" %
%   I:3.0/11  PE4  "Bin Clear" %
%   B3:5/8  "In Auto One Shot Flag" %
% Rung: 14 %
SOR BST XIC O:0.0/11 XIO O:5.0/13 NXB XIO O:0.0/11 XIC I:3.0/4 BND OTE O:5.0/14 EOR
%   O:0.0/11  IND_STACKER_AUTO %
%   O:5.0/13  BIN_STOP_DOWN %
%   I:3.0/4  "SEL STACK BIN STOP UP" %
%   O:5.0/14  BIN_STOP_UP %
% Rung: 15 %
SOR BST XIC O:0.0/11 BST XIO I:3.0/11 XIC I:3.0/9 NXB XIC O:5.0/13 BND BST XIC B3:5/4 NXB XIC I:3.0/11 BND NXB XIO O:0.0/11 XIC I:3.0/5 BND OTE O:5.0/13 EOR
%   O:0.0/11  IND_STACKER_AUTO %
%   I:3.0/11  PE4  "Bin Clear" %
%   I:3.0/9  PE2  "STACKER BIN IN" %
%   O:5.0/13  BIN_STOP_DOWN %
%   B3:5/4  "Stacker Bin Stop Drop Flag" %
%   I:3.0/5  "SEL STACK BIN STOP DOWN" %

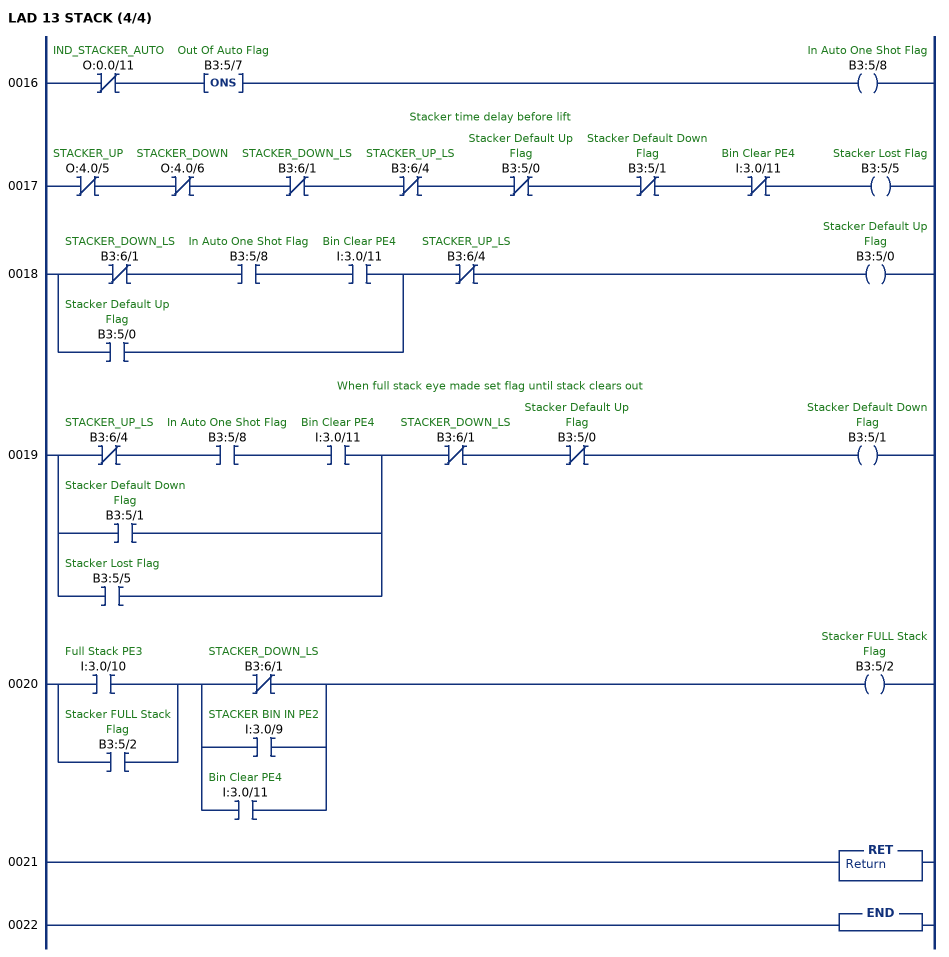
% Rung: 16 %
SOR XIO O:0.0/11 ONS B3:5/7 OTE B3:5/8 EOR
%   O:0.0/11  IND_STACKER_AUTO %
%   B3:5/7  "Out Of Auto Flag" %
%   B3:5/8  "In Auto One Shot Flag" %
% Rung: 17 %
% Stacker time delay before lift %
SOR XIO O:4.0/5 XIO O:4.0/6 XIO B3:6/1 XIO B3:6/4 XIO B3:5/0 XIO B3:5/1 XIO I:3.0/11 OTE B3:5/5 EOR
%   O:4.0/5  STACKER_UP %
%   O:4.0/6  STACKER_DOWN %
%   B3:6/1  STACKER_DOWN_LS %
%   B3:6/4  STACKER_UP_LS %
%   B3:5/0  "Stacker Default Up Flag" %
%   B3:5/1  "Stacker Default Down Flag" %
%   I:3.0/11  PE4  "Bin Clear" %
%   B3:5/5  "Stacker Lost Flag" %
% Rung: 18 %
SOR BST XIO B3:6/1 XIC B3:5/8 XIC I:3.0/11 NXB XIC B3:5/0 BND XIO B3:6/4 OTE B3:5/0 EOR
%   B3:6/1  STACKER_DOWN_LS %
%   B3:5/8  "In Auto One Shot Flag" %
%   I:3.0/11  PE4  "Bin Clear" %
%   B3:5/0  "Stacker Default Up Flag" %
%   B3:6/4  STACKER_UP_LS %
% Rung: 19 %
% When full stack eye made set flag until stack clears out %
SOR BST XIO B3:6/4 XIC B3:5/8 XIC I:3.0/11 NXB XIC B3:5/1 NXB XIC B3:5/5 BND XIO B3:6/1 XIO B3:5/0 OTE B3:5/1 EOR
%   B3:6/4  STACKER_UP_LS %
%   B3:5/8  "In Auto One Shot Flag" %
%   I:3.0/11  PE4  "Bin Clear" %
%   B3:5/1  "Stacker Default Down Flag" %
%   B3:5/5  "Stacker Lost Flag" %
%   B3:6/1  STACKER_DOWN_LS %
%   B3:5/0  "Stacker Default Up Flag" %
% Rung: 20 %
SOR BST XIC I:3.0/10 NXB XIC B3:5/2 BND BST XIO B3:6/1 NXB BST XIC I:3.0/9 NXB XIC I:3.0/11 BND BND OTE B3:5/2 EOR
%   I:3.0/10  PE3  "Full Stack" %
%   B3:5/2  "Stacker FULL Stack Flag" %
%   B3:6/1  STACKER_DOWN_LS %
%   I:3.0/9  PE2  "STACKER BIN IN" %
%   I:3.0/11  PE4  "Bin Clear" %
% Rung: 21 %
SOR RET EOR
% Rung: 22 %
SOR END EOR

OTHER DOCUMENTED ADDRESSES
  B3:0/9  SANITIZE_LTCH  "Triggered by reset limit sw."
  B3:0/10  SANITIZE_BIT  "Allow crdl ltch2 to unlatch only once until sanitize cycle is over"
  B3:0/11  CRDL_EN  "mcr on and no encoder fault"
  B3:0/15  CRDL_HAND_SS
  B3:1/1  RINSE_SELECT  "Turn ON Rinse"
  B3:2/13  SHOW_INPUTS_OUTPUTS  "HMI"
  B3:3/3  "Conveyor Transition"
  B3:3/4  "HMI"
  B3:3/10  BIN_ON_BYPASS
  B3:5/13  TEST
  C5:0/CU  EVENT_COUNTER
  I:0.4/0  DESTACK_LINER
  I:0.5/0  STACKER_LINEAR
  L10:1/1  FAULT_MESSAGES
  N7:1/0  "Fault-Infeed Blocked"
  N7:1/1  "Fault-Outfeed Blocked"
  N7:1/2  "Fault-Cradle Overtravel Up"
  N7:1/3  "Fault-Cradle Overtravel down"
  N7:1/4  "Fault-Torque Cradle Inverter"
  N7:1/5  "Main Tank Low"
  N7:1/6  "Encoder Fault"
  N7:1/7  "Fill Main Tank"
  N7:7  LOWER_WASH_TURN_OFF
  N9:0  K1
  O:0.0/7  NOT_USED
  O:2.0/1  RINSE_SOLENOID  "Rinse after wash"
  O:5.0/9  OPTIONAL_RINSE
  T4:0/EN  CRDL_DWN_T  "Allows cradle to set down completely before conv starts"
  T4:1  CRDL_FLT_T1
  T4:2  CRDL_FLT_T2
  T4:6  SANITIZE_T
  T4:7  CRDL_DWN_T2  "Inhibits cradle up for 5 sec. after cradle sets down"
  T4:10  CRADLE_TIMER  "Cradle travel watch dog timer"

COMMENTS NOT ATTACHED TO A CURRENT RUNG
  N7:1/0: As long as the bit is set, the message will be displayed.  Bit #1 is Message #1.  Bit #3 is message #4.  Binary to decimal.
  T4:6.PRE: As long as the bit is set, the message will be displayed.  Bit #1 is Message #1.  Bit #3 is message #4.  Binary to decimal.
  T4:7: Timer not used
  N7:26: CALCULATE SLOW PICK UP SP
  N7:23: CALCULATE LIFT SET POINT
  N7:28: CALCULATE LIFT SET POINT

REVISION NOTES
  0: Added barrier and overtravel tatches
  1: Added indepentent barrier and overtravel catches
  2: Changed ffrom Panel #8.  Added B3:0/1 to prevent B3:0/5 from latching up while cradle is not down
  3: Added more troubleshooting help - step sequences
  4: Costa Rica Panel #19 with individual upper and lower wash solenoids
  5: Changed to 1400 with additional input and output cards

DATA TABLE (non-zero values as saved)
DATA B3
% B3:0 % 0X5D02 0X4003 0X0830 0X0400 0X0011 0X0082 0X0018
DATA T4
% .PRE .ACC %
% T4:0 % 50 50
% T4:1 % 1 0
% T4:2 % 1 0
% T4:3 % 500 0
% T4:4 % 2 2
% T4:5 % 5 5
% T4:6 % 658 0
% T4:7 % 375 500
% T4:8 % 5 0
% T4:9 % 2 0
% T4:10 % 500 0
% T4:11 % 75 0
% T4:12 % 150 0
% T4:13 % 180 0
% T4:14 % 180 0
% T4:15 % 500 0
% T4:16 % 500 0
% T4:17 % 100 0
% T4:18 % 100 0
% T4:20 % 7 0
% T4:21 % 625 0
% T4:22 % 270 0
% T4:23 % 69 0
% T4:24 % 69 0
% T4:25 % 6 0
% T4:26 % 70 0
% T4:27 % 75 0
% T4:28 % 400 0
% T4:30 % 50 100
% T4:31 % 50 0
% T4:32 % 1 0
% T4:33 % 1 0
% T4:34 % 25 0
% T4:35 % 100 0
% T4:36 % 100 0
% T4:37 % 6 0
DATA N7
% N7:0 % 86 0 10 65 130 21 24 0 69 0
% N7:10 % 9 9 0 0 0 0 0 0 0 0
DATA F8
% F8:0 % 88 0 0 0 0
% F8:5 % 4077 115.61 35.26511 0 0
% F8:20 % 0.125 0.5 7.25 7.75 7.25
% F8:25 % 27.85 35.1 0 0 35.375
